// TwinCAT 3 PLC project reactor
// ProgramVersion: 3.1.4023.0
// libraries:
//   Tc2_DataExchange, * (Beckhoff Automation GmbH)
//   Tc2_Standard, * (Beckhoff Automation GmbH)
//   Tc2_System, * (Beckhoff Automation GmbH)
//   Tc3_Module, * (Beckhoff Automation GmbH)
// project tree:
//   FB/ FB_ReadAmsValue.TcPOU, FB_WriteAmsValue.TcPOU
//   GVLs/ GVL.TcGVL, SUPVams.TcGVL
//   / PlcTask.TcTTO
//   POUs/ MAIN.TcPOU, POU_readSupvData.TcPOU, POU_writeReactorToSupvData.TcPOU
// real-time tasks:
//   TASK PlcTask: cycle T#10ms, priority 20, ADS port 350

CONFIGURATION reactor
    RESOURCE PLC ON TwinCAT3
        TASK PlcTask(INTERVAL := T#10ms, PRIORITY := 20);
        PROGRAM MAIN WITH PlcTask : MAIN;
    END_RESOURCE
END_CONFIGURATION

// ---- GVLs/GVL.TcGVL
{attribute 'qualified_only'}
VAR_GLOBAL
	// setpoints
	PROD_RATE_SP					:	LREAL	:= 0.0;	// production rate 
	L_STRIPPER_SP					:	LREAL	:= 0.0;	// stripper level
	L_SEPARATOR_SP					:	LREAL	:= 0.0;	// separator level
	L_REACTOR_SP					:	LREAL	:= 0.0;	// reactor level
	P_REACTOR_SP					:	LREAL;	// reactor pressure
	PCT_G_SP						:	LREAL;	// Mole percent G
	YA_SP							: 	LREAL;	// yA 
	YAC_SP							:	LREAL;	// yAC
	T_REACTOR_SP					:	LREAL;	// reactor temperature
	RECYC_VALVE_SP					:	LREAL;	// Recycle valve position
	STEAM_VALVE_SP					:	LREAL;	// Steam valve position
	L_AGITATOR_SP					:	LREAL;	// agitator setting		
	
	// Intermediate values
	Fp							:	LREAL; 	

	// actual production metrics
	COST						:	LREAL :=0.0;
	PctG						:	LREAL :=0.0;

	// process variables
	XMEAS						:	ARRAY[1..41] OF LREAL;
	XMEAS_TO_SUPV				:	ARRAY[1..10] OF LREAL;
	XMV							:	ARRAY[1..12] OF LREAL;
	XMV_TO_SUPV					:	ARRAY[1..5] OF LREAL;
	
	// intermediate variables
	SEP_TEMP_SP					:	LREAL;	// separator temperaure setpoint
	RI							:	ARRAY[1..6] OF LREAL;	// ratio trimming outputs
	EADJ						:	LREAL;	// adjustment to production rate
	PCTG_SP						:	LREAL;	// setpoint for precent G
	
	// shutdown indicator
	SD_FLAG						: 	BOOL	:= FALSE;

	// operating time
	OPTIME					:	LREAL := 0.0;	
	
END_VAR

// ---- GVLs/SUPVams.TcGVL
{attribute 'qualified_only'}
VAR_GLOBAL
	sNetId: T_AmsNetId := '5.30.23.91.1.1';
	nPort: T_AmsPort := 851;	
END_VAR

// ---- POUs/MAIN.TcPOU
PROGRAM MAIN
VAR

END_VAR

POU_readSupvData();
POU_writeReactorToSupvData();

END_PROGRAM

// ---- POUs/POU_readSupvData.TcPOU
PROGRAM POU_readSupvData
VAR
	sNetId: T_AmsNetId := SUPVams.sNetId;	// '5.30.23.91.1.1';
	nPort: T_AmsPort := SUPVams.nPort; 		// 851
	FB_ReadAmsValue_Fp: FB_ReadAmsValue;
	FB_ReadAmsValue_R2: FB_ReadAmsValue;
	FB_ReadAmsValue_R3: FB_ReadAmsValue;
	FB_ReadAmsValue_TReactor: FB_ReadAmsValue;
	FB_ReadAmsValue_YA: FB_ReadAmsValue;
	FB_ReadAmsValue_YAC: FB_ReadAmsValue;
	FB_ReadAmsValue_AGI: FB_ReadAmsValue;
END_VAR

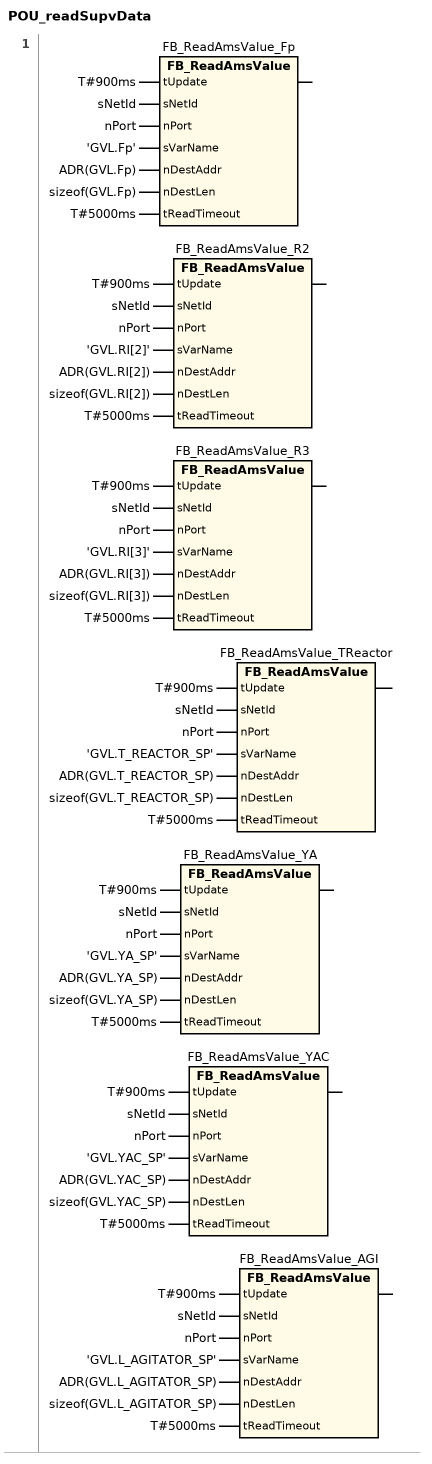
// NETWORK 1
FB_ReadAmsValue_Fp(
    tUpdate := T#900ms,
    sNetId := sNetId,
    nPort := nPort,
    sVarName := 'GVL.Fp',
    nDestAddr := ADR(GVL.Fp),
    nDestLen := sizeof(GVL.Fp),
    tReadTimeout := T#5000ms); // FB_ReadAmsValue
FB_ReadAmsValue_R2(
    tUpdate := T#900ms,
    sNetId := sNetId,
    nPort := nPort,
    sVarName := 'GVL.RI[2]',
    nDestAddr := ADR(GVL.RI[2]),
    nDestLen := sizeof(GVL.RI[2]),
    tReadTimeout := T#5000ms); // FB_ReadAmsValue
FB_ReadAmsValue_R3(
    tUpdate := T#900ms,
    sNetId := sNetId,
    nPort := nPort,
    sVarName := 'GVL.RI[3]',
    nDestAddr := ADR(GVL.RI[3]),
    nDestLen := sizeof(GVL.RI[3]),
    tReadTimeout := T#5000ms); // FB_ReadAmsValue
FB_ReadAmsValue_TReactor(
    tUpdate := T#900ms,
    sNetId := sNetId,
    nPort := nPort,
    sVarName := 'GVL.T_REACTOR_SP',
    nDestAddr := ADR(GVL.T_REACTOR_SP),
    nDestLen := sizeof(GVL.T_REACTOR_SP),
    tReadTimeout := T#5000ms); // FB_ReadAmsValue
FB_ReadAmsValue_YA(
    tUpdate := T#900ms,
    sNetId := sNetId,
    nPort := nPort,
    sVarName := 'GVL.YA_SP',
    nDestAddr := ADR(GVL.YA_SP),
    nDestLen := sizeof(GVL.YA_SP),
    tReadTimeout := T#5000ms); // FB_ReadAmsValue
FB_ReadAmsValue_YAC(
    tUpdate := T#900ms,
    sNetId := sNetId,
    nPort := nPort,
    sVarName := 'GVL.YAC_SP',
    nDestAddr := ADR(GVL.YAC_SP),
    nDestLen := sizeof(GVL.YAC_SP),
    tReadTimeout := T#5000ms); // FB_ReadAmsValue
FB_ReadAmsValue_AGI(
    tUpdate := T#900ms,
    sNetId := sNetId,
    nPort := nPort,
    sVarName := 'GVL.L_AGITATOR_SP',
    nDestAddr := ADR(GVL.L_AGITATOR_SP),
    nDestLen := sizeof(GVL.L_AGITATOR_SP),
    tReadTimeout := T#5000ms); // FB_ReadAmsValue

END_PROGRAM

// ---- FB/FB_ReadAmsValue.TcPOU
FUNCTION_BLOCK FB_ReadAmsValue
VAR_INPUT
	tUpdate					:	TIME 				:=T#900MS;
	
	sNetId					:	T_AmsNetId			:='';
	nPort					:	T_AmsPort			:=851;
	sVarName				:	STRING(255)			:='';
	nDestAddr				:	PVOID;
	nDestLen				:	UDINT;
	tReadTimeout			:	TIME				:=T#2000MS;
	
END_VAR

VAR_OUTPUT
END_VAR

VAR
	
	bReadError		: BOOL := FALSE;
	nReadErrorId	: UDINT;
	PT_Read			: TIME := T#5S;
	
	ET_Read			: TIME := T#0MS;
	bReadEnable		: BOOL := FALSE;
	readBusy		: BOOL := FALSE;
	
	TON_Read		: TON;
	fb_reader	: FB_ReadAdsSymByName;
END_VAR

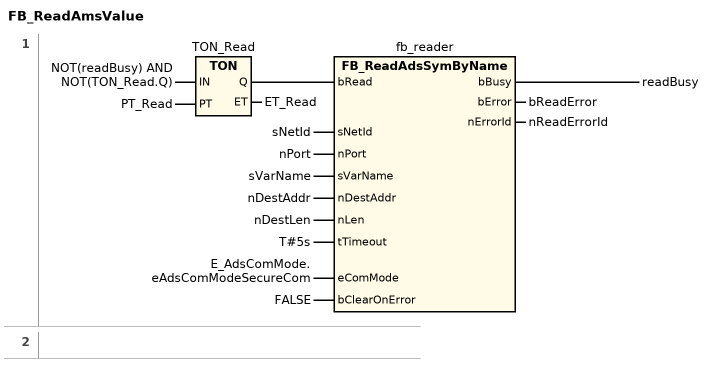
// NETWORK 1
TON_Read(IN := NOT(readBusy) AND NOT(TON_Read.Q), PT := PT_Read, ET => ET_Read); // TON
fb_reader(
    bRead := TON_Read.Q,
    sNetId := sNetId,
    nPort := nPort,
    sVarName := sVarName,
    nDestAddr := nDestAddr,
    nLen := nDestLen,
    tTimeout := T#5s,
    eComMode := E_AdsComMode.eAdsComModeSecureCom,
    bClearOnError := FALSE,
    bError => bReadError,
    nErrorId => nReadErrorId); // FB_ReadAdsSymByName
readBusy := fb_reader.bBusy;

// NETWORK 2

END_FUNCTION_BLOCK

// ---- POUs/POU_writeReactorToSupvData.TcPOU
PROGRAM POU_writeReactorToSupvData
VAR
	sNetId: T_AmsNetId := SUPVams.sNetId;	// '5.30.23.91.1.1';
	nPort: T_AmsPort := SUPVams.nPort; 		// 851	

	FB_WriteAmsValue_XMEAS: FB_WriteAmsValue;
END_VAR

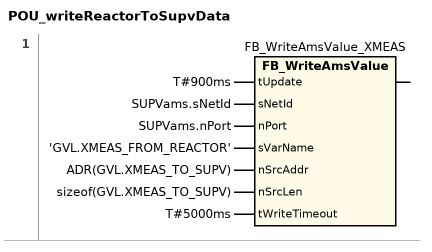
// NETWORK 1
FB_WriteAmsValue_XMEAS(
    tUpdate := T#900ms,
    sNetId := SUPVams.sNetId,
    nPort := SUPVams.nPort,
    sVarName := 'GVL.XMEAS_FROM_REACTOR',
    nSrcAddr := ADR(GVL.XMEAS_TO_SUPV),
    nSrcLen := sizeof(GVL.XMEAS_TO_SUPV),
    tWriteTimeout := T#5000ms); // FB_WriteAmsValue

END_PROGRAM

// ---- FB/FB_WriteAmsValue.TcPOU
FUNCTION_BLOCK FB_WriteAmsValue
VAR_INPUT
	tUpdate					:	TIME 				:=T#900MS;
	
	sNetId					:	T_AmsNetId			:='';
	nPort					:	T_AmsPort			:=851;
	sVarName				:	STRING(255)			:='';
	nSrcAddr				:	PVOID;
	nSrcLen					:	UDINT;
	tWriteTimeout			:	TIME				:=T#2000MS;
	
END_VAR

VAR_OUTPUT
END_VAR

VAR
	
	bWriteError			: BOOL := FALSE;
	nWriteErrorId		: UDINT;
	PT_Write			: TIME := T#5S;
	
	ET_Write			: TIME := T#0MS;
	bReadEnable			: BOOL := FALSE;
	bWriteBusy			: BOOL := FALSE;
	
	TON_Write		: TON;
	FB_writer		: FB_WriteAdsSymByName;
END_VAR

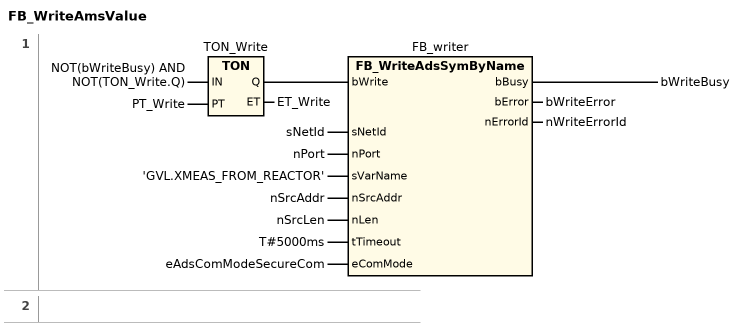
// NETWORK 1
TON_Write(IN := NOT(bWriteBusy) AND NOT(TON_Write.Q), PT := PT_Write, ET => ET_Write); // TON
FB_writer(
    bWrite := TON_Write.Q,
    sNetId := sNetId,
    nPort := nPort,
    sVarName := 'GVL.XMEAS_FROM_REACTOR',
    nSrcAddr := nSrcAddr,
    nLen := nSrcLen,
    tTimeout := T#5000ms,
    eComMode := eAdsComModeSecureCom,
    bError => bWriteError,
    nErrorId => nWriteErrorId); // FB_WriteAdsSymByName
bWriteBusy := FB_writer.bBusy;

// NETWORK 2

END_FUNCTION_BLOCK
